(* IEC 61131-3 sources: CodesysTest/alpha/export/Pro18_1174_04.dev/Plc Logic/Application/Motors/Festo/FB_FestoMotor.pou, 1 file *)

(* ---- InitDrive.m.st ---- *)
(*#-#-#-#-#-#-#-#-#-#---Declaration---#-#-#-#-#-#-#-#-#-#-#-#-#*)

METHOD PRIVATE InitDrive
VAR_INPUT
END_VAR
(*#-#-#-#-#-#-#-#-#-#---Implementation---#-#-#-#-#-#-#-#-#-#-#-#-#*)

//Initialize the drive to prepare for a move
CRTL_Axis.EnableDrive := TRUE;
CRTL_Axis.Halt := TRUE;
CRTL_Axis.Stop := TRUE;
//CRTL_Axis.StartTask := FALSE;
commandSuccessful := FALSE;
